# EPICS autosave request: ADApp/Db/NDPluginBase_settings.req
$(P)$(R)NDArrayPort
$(P)$(R)NDArrayAddress
$(P)$(R)EnableCallbacks
$(P)$(R)MemoryPoolDiagScan.SCAN
$(P)$(R)MinCallbackTime
$(P)$(R)BlockingCallbacks
$(P)$(R)QueueSize
$(P)$(R)NumThreads
$(P)$(R)SortTime
$(P)$(R)SortMode
$(P)$(R)SortSize
file "NDArrayBase_settings.req", P=$(P), R=$(R)
$(P)$(R)NDAttributesFile
$(P)$(R)ArrayCounter_RBV.TSE
$(P)$(R)EpicsTSNsec_RBV.TSE
$(P)$(R)EpicsTSSec_RBV.TSE
$(P)$(R)UniqueId_RBV.TSE
$(P)$(R)TimeStamp_RBV.TSE
